// TIA Portal V16 export
// export: Created 2021-11-12T13:31:56.937165Z, ExportSetting WithDefaults, DisplayName Totally Integrated Automation Portal, DisplayVersion V16 Update 3, DisplayName TIA Portal Version Control Interface, DisplayVersion V16 Update 2, DisplayName TIA Portal Openness, DisplayVersion V16 Update 3, DisplayName SINAMICS Startdrive Advanced, DisplayVersion V16 Update 5, DisplayName SINAMICS Startdrive G130, G150, S120, S150, SINAMICS MV, S210, DisplayVersion V16 Update 5, DisplayName SINAMICS Startdrive G110M, G120, G120C, G120D, G120P, G115D, DisplayVersion V16 Update 5, DisplayName STEP 7 Professional, DisplayVersion V16 Update 3, DisplayName STEP 7 Safety, DisplayVersion V16, DisplayName WinCC UA Professional, DisplayVersion V16 Update 3
DATA_BLOCK "HMI_PARAM_000+UC20"   // DB183
{ S7_Optimized_Access := 'TRUE' }
VERSION : 0.1
// stored: AutoNumber true, DBAccessibleFromOPCUA true, IsOnlyStoredInLoadMemory false, IsRetainMemResEnabled false, IsWriteProtectedInAS false, MemoryReserve 100
   VAR
      xxxxx___BinarySensors___xxxxx : Byte;
      xxxxx___BinaryOthers___xxxxx : Byte;
      FB21_14 { S7_SetPoint := 'True'} : "UDT_CH_DI_Parameter";   // 230V Osvětlení rozvaděče se zásuvkou je OK
      FC21_14 { S7_SetPoint := 'True'} : "UDT_CH_DI_Parameter";   // 230V Chlazeni rozvaděče je OK
      EC01_3 { S7_SetPoint := 'True'} : "UDT_CH_DI_Parameter";   // Chlazení rozvaděče je OK
      FC01_14 { S7_SetPoint := 'True'} : "UDT_CH_DI_Parameter";   // 400V Napájení 24V DC je OK
      TB01_14 { S7_SetPoint := 'True'} : "UDT_CH_DI_Parameter";   // Napájení 24V DC je OK
      FC30_14 { S7_SetPoint := 'True'} : "UDT_CH_DI_Parameter";   // 24V Distribuce je OK
      FC30_24 { S7_SetPoint := 'True'} : "UDT_CH_DI_Parameter";   // 24V Distribuce 90 >% zatížení
      FC50_14 : "UDT_CH_DI_Parameter";   // 24V Distribuce je OK
      FC50_24 : "UDT_CH_DI_Parameter";   // 24V Distribuce 90 >% zatížení
      xxxxx___AnalogueSensors___xxxxx : Byte;
      xxxxx___Drives___xxxxx : Byte;
      xxxxx___Other___xxxxx : Byte;
      xxxxx___Alarms___xxxxx : Byte;
      FB21_15 { S7_SetPoint := 'True'} : "UDT_DI_Mon_Parameter";   // 230V Osvětlení rozvaděče se zásuvkou je OK
      FC21_15 { S7_SetPoint := 'True'} : "UDT_DI_Mon_Parameter";   // 230V Chlazeni rozvaděče je OK
      EC01_4 { S7_SetPoint := 'True'} : "UDT_DI_Mon_Parameter";   // Chlazení rozvaděče je OK
      FC01_15 { S7_SetPoint := 'True'} : "UDT_DI_Mon_Parameter";   // 400V Napájení 24V DC je OK
      TB01_15 { S7_SetPoint := 'True'} : "UDT_DI_Mon_Parameter";   // Napájení 24V DC je OK
      FC30_15 { S7_SetPoint := 'True'} : "UDT_DI_Mon_Parameter";   // 24V Distribuce je OK
      FC30_25 { S7_SetPoint := 'True'} : "UDT_DI_Mon_Parameter";   // 24V Distribuce 90 >% zatížení
      FC50_15 : "UDT_DI_Mon_Parameter";   // 24V Distribuce je OK
      FC50_25 : "UDT_DI_Mon_Parameter";   // 24V Distribuce 90 >% zatížení
   END_VAR
BEGIN
END_DATA_BLOCK
